Fanuc TP program (LS listing): tool_3_dropoff_aproach.ls

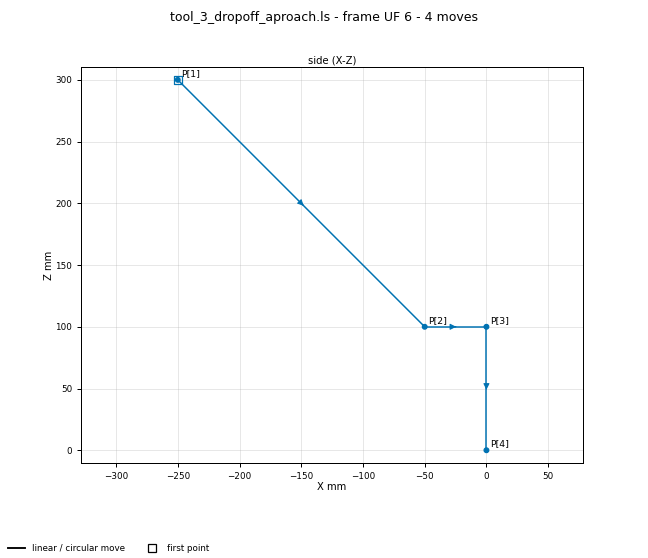
[picture p0: tool path of tool_3_dropoff_aproach.ls in frame UF 6, 4 of 4 moves have a stored position in this frame; points joined in program order, loops and branches not executed]
/PROG  TOOL_3_DROPOFF_APROACH
/ATTR
OWNER		= MNEDITOR;
COMMENT		= "";
PROG_SIZE	= 911;
CREATE		= DATE 21-04-28  TIME 16:59:04;
MODIFIED	= DATE 22-03-01  TIME 07:31:20;
FILE_NAME	= ;
VERSION		= 0;
LINE_COUNT	= 13;
MEMORY_SIZE	= 1239;
PROTECT		= READ_WRITE;
TCD:  STACK_SIZE	= 0,
      TASK_PRIORITY	= 50,
      TIME_SLICE	= 0,
      BUSY_LAMP_OFF	= 0,
      ABORT_REQUEST	= 0,
      PAUSE_REQUEST	= 0;
DEFAULT_GROUP	= 1,*,*,*,*;
CONTROL_CODE	= 00000000 00000000;
/APPL

AUTO_SINGULARITY_HEADER;
  ENABLE_SINGULARITY_AVOIDANCE   : TRUE;
/MN
   1:  UFRAME_NUM=6 ;
   2:  UTOOL_NUM=2 ;
   3:  !MOVE TO FLIGHT HEIGHT (x axis) ;
   4:L P[1] 100mm/sec FINE ACC10    ;
   5:  !LOWER TO SAFE OFFSET ;
   6:L P[2] 100mm/sec FINE ACC10    ;
   7:  !MOVE OVER PRONGS ;
   8:L P[3] 100mm/sec FINE ACC10    ;
   9:  !ENGAGE TOOL ONTO PRONG (origin) ;
  10:L P[4] 100mm/sec FINE ACC10    ;
  11:  WAIT   1.00(sec) ;
  12:  !PLC TOOL UNLOCK ;
  13:  CALL PLCHANDSHAKE    ;
/POS
P[1]{
   GP1:
	UF : 6, UT : 2,		CONFIG : 'F U T, 0, 0, 0',
	X =  -250.000  mm,	Y =     0.000  mm,	Z =   300.000  mm,
	W =     0.000 deg,	P =     0.000 deg,	R =     0.000 deg,
	E1= -1290.487  mm
};
P[2]{
   GP1:
	UF : 6, UT : 2,		CONFIG : 'F U T, 0, 0, 0',
	X =   -50.000  mm,	Y =    -2.043  mm,	Z =   100.000  mm,
	W =     0.000 deg,	P =     0.000 deg,	R =     0.000 deg,
	E1= -1290.487  mm
};
P[3]{
   GP1:
	UF : 6, UT : 2,		CONFIG : 'F U T, 0, 0, 0',
	X =     0.000  mm,	Y =    -2.043  mm,	Z =   100.000  mm,
	W =     0.000 deg,	P =     0.000 deg,	R =     0.000 deg,
	E1= -1290.487  mm
};
P[4]{
   GP1:
	UF : 6, UT : 2,		CONFIG : 'F U T, 0, 0, 0',
	X =     0.000  mm,	Y =    -2.043  mm,	Z =     0.000  mm,
	W =     0.000 deg,	P =     0.000 deg,	R =     0.000 deg,
	E1= -1290.487  mm
};
/END
